TYPE ST_AteqIo :
STRUCT
	stRead  : ST_AteqRead;
    stWrite : ST_AteqWrite;
END_STRUCT
END_TYPE

(* stored: Version 1.1.0.1
   DUT ST_AteqIo: Id {7ce7ac0c-1c92-4cec-a3bd-bf1f5c9de48e} *)
